{attribute 'GeneratedUsingTerminal: KL9110'}
{attribute addProperty BoxType "KL9110"}
{attribute addProperty Id "PowerAT %I*BOOL0ShortCircuitAT %I*BOOL0"}
{attribute addProperty CRC "1688914119"}
{attribute addProperty Size "0"}
TYPE Channel_64AAC8C7 EXTENDS InputBase_8311D824 :
STRUCT
	{attribute addProperty Name "Power"}
	Power AT %I* : BOOL;
	{attribute addProperty Name "ShortCircuit"}
	ShortCircuit AT %I* : BOOL;
END_STRUCT
END_TYPE

(* stored: Version 1.2.0.0, ProductVersion 3.1.4024.11
   DUT Channel_64AAC8C7: Id {51341d68-32f8-4570-ad90-8c8da0da5406} *)
